// TIA Portal V20 export
FUNCTION_BLOCK "Simulation"   // FB50062, LAD
// stored: MemoryReserve 100, Namespace Unit1.Em7, SetENOAutomatically false
   VAR_INPUT
      simulation { ExternalAccessible := 'False'; ExternalVisible := 'False'; ExternalWritable := 'False'} : Bool;
   END_VAR
   VAR
      instActuator { ExternalAccessible := 'False'; ExternalVisible := 'False'; ExternalWritable := 'False'} : Array[0..19] of "LER_SimActuator";
   END_VAR
   VAR_TEMP   // added for the SCL form of the ladder/FBD networks
      _w1 : Bool;
      _w2 : Bool;
      _w3 : Bool;
      _w4 : Bool;
      _w5 : Bool;
      _w6 : Bool;
   END_VAR
BEGIN

REGION Network 1: Two Way Actuator
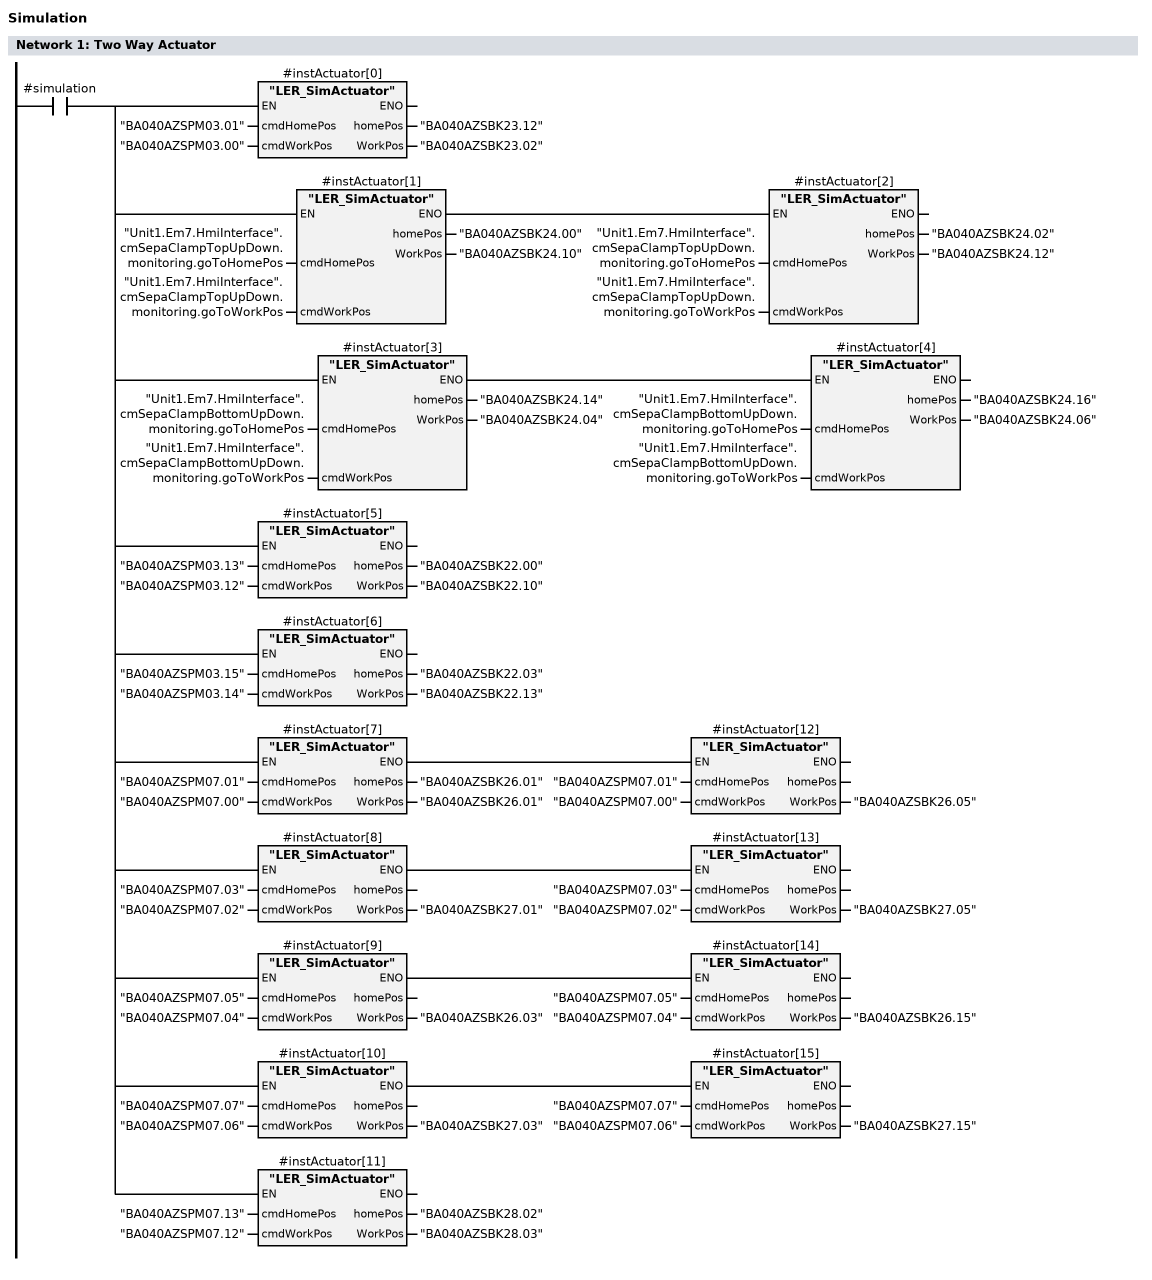
   RUNG wire#powerrail
      Contact( #simulation )
      wire#w1
      #instActuator[0](cmdHomePos := "BA040AZSPM03.01", cmdWorkPos := "BA040AZSPM03.00", homePos => "BA040AZSBK23.12", WorkPos => "BA040AZSBK23.02")
   END_RUNG
   RUNG wire#w1
      #instActuator[1](cmdHomePos := "Unit1.Em7.HmiInterface".cmSepaClampTopUpDown.monitoring.goToHomePos, cmdWorkPos := "Unit1.Em7.HmiInterface".cmSepaClampTopUpDown.monitoring.goToWorkPos, homePos => "BA040AZSBK24.00", WorkPos => "BA040AZSBK24.10")
      #instActuator[2](cmdHomePos := "Unit1.Em7.HmiInterface".cmSepaClampTopUpDown.monitoring.goToHomePos, cmdWorkPos := "Unit1.Em7.HmiInterface".cmSepaClampTopUpDown.monitoring.goToWorkPos, homePos => "BA040AZSBK24.02", WorkPos => "BA040AZSBK24.12")
   END_RUNG
   RUNG wire#w1
      #instActuator[3](cmdHomePos := "Unit1.Em7.HmiInterface".cmSepaClampBottomUpDown.monitoring.goToHomePos, cmdWorkPos := "Unit1.Em7.HmiInterface".cmSepaClampBottomUpDown.monitoring.goToWorkPos, homePos => "BA040AZSBK24.14", WorkPos => "BA040AZSBK24.04")
      #instActuator[4](cmdHomePos := "Unit1.Em7.HmiInterface".cmSepaClampBottomUpDown.monitoring.goToHomePos, cmdWorkPos := "Unit1.Em7.HmiInterface".cmSepaClampBottomUpDown.monitoring.goToWorkPos, homePos => "BA040AZSBK24.16", WorkPos => "BA040AZSBK24.06")
   END_RUNG
   RUNG wire#w1
      #instActuator[5](cmdHomePos := "BA040AZSPM03.13", cmdWorkPos := "BA040AZSPM03.12", homePos => "BA040AZSBK22.00", WorkPos => "BA040AZSBK22.10")
   END_RUNG
   RUNG wire#w1
      #instActuator[6](cmdHomePos := "BA040AZSPM03.15", cmdWorkPos := "BA040AZSPM03.14", homePos => "BA040AZSBK22.03", WorkPos => "BA040AZSBK22.13")
   END_RUNG
   RUNG wire#w1
      #instActuator[7](cmdHomePos := "BA040AZSPM07.01", cmdWorkPos := "BA040AZSPM07.00", homePos => "BA040AZSBK26.01", WorkPos => "BA040AZSBK26.01")
      #instActuator[12](cmdHomePos := "BA040AZSPM07.01", cmdWorkPos := "BA040AZSPM07.00", homePos =>, WorkPos => "BA040AZSBK26.05")
   END_RUNG
   RUNG wire#w1
      #instActuator[8](cmdHomePos := "BA040AZSPM07.03", cmdWorkPos := "BA040AZSPM07.02", homePos =>, WorkPos => "BA040AZSBK27.01")
      #instActuator[13](cmdHomePos := "BA040AZSPM07.03", cmdWorkPos := "BA040AZSPM07.02", homePos =>, WorkPos => "BA040AZSBK27.05")
   END_RUNG
   RUNG wire#w1
      #instActuator[9](cmdHomePos := "BA040AZSPM07.05", cmdWorkPos := "BA040AZSPM07.04", homePos =>, WorkPos => "BA040AZSBK26.03")
      #instActuator[14](cmdHomePos := "BA040AZSPM07.05", cmdWorkPos := "BA040AZSPM07.04", homePos =>, WorkPos => "BA040AZSBK26.15")
   END_RUNG
   RUNG wire#w1
      #instActuator[10](cmdHomePos := "BA040AZSPM07.07", cmdWorkPos := "BA040AZSPM07.06", homePos =>, WorkPos => "BA040AZSBK27.03")
      #instActuator[15](cmdHomePos := "BA040AZSPM07.07", cmdWorkPos := "BA040AZSPM07.06", homePos =>, WorkPos => "BA040AZSBK27.15")
   END_RUNG
   RUNG wire#w1
      #instActuator[11](cmdHomePos := "BA040AZSPM07.13", cmdWorkPos := "BA040AZSPM07.12", homePos => "BA040AZSBK28.02", WorkPos => "BA040AZSBK28.03")
   END_RUNG
   // the same network as SCL:
   IF #simulation THEN
       #instActuator[0](cmdHomePos := "BA040AZSPM03.01",   // "LER_SimActuator"
                        cmdWorkPos := "BA040AZSPM03.00",
                        homePos => "BA040AZSBK23.12",
                        WorkPos => "BA040AZSBK23.02");
   END_IF;
   #instActuator[1](EN := #simulation,   // "LER_SimActuator"
                    cmdHomePos := "Unit1.Em7.HmiInterface".cmSepaClampTopUpDown.monitoring.goToHomePos,
                    cmdWorkPos := "Unit1.Em7.HmiInterface".cmSepaClampTopUpDown.monitoring.goToWorkPos,
                    homePos => "BA040AZSBK24.00",
                    WorkPos => "BA040AZSBK24.10",
                    ENO => #_w1);
   IF #_w1 THEN
       #instActuator[2](cmdHomePos := "Unit1.Em7.HmiInterface".cmSepaClampTopUpDown.monitoring.goToHomePos,   // "LER_SimActuator"
                        cmdWorkPos := "Unit1.Em7.HmiInterface".cmSepaClampTopUpDown.monitoring.goToWorkPos,
                        homePos => "BA040AZSBK24.02",
                        WorkPos => "BA040AZSBK24.12");
   END_IF;
   #instActuator[3](EN := #simulation,   // "LER_SimActuator"
                    cmdHomePos := "Unit1.Em7.HmiInterface".cmSepaClampBottomUpDown.monitoring.goToHomePos,
                    cmdWorkPos := "Unit1.Em7.HmiInterface".cmSepaClampBottomUpDown.monitoring.goToWorkPos,
                    homePos => "BA040AZSBK24.14",
                    WorkPos => "BA040AZSBK24.04",
                    ENO => #_w2);
   IF #_w2 THEN
       #instActuator[4](cmdHomePos := "Unit1.Em7.HmiInterface".cmSepaClampBottomUpDown.monitoring.goToHomePos,   // "LER_SimActuator"
                        cmdWorkPos := "Unit1.Em7.HmiInterface".cmSepaClampBottomUpDown.monitoring.goToWorkPos,
                        homePos => "BA040AZSBK24.16",
                        WorkPos => "BA040AZSBK24.06");
   END_IF;
   IF #simulation THEN
       #instActuator[5](cmdHomePos := "BA040AZSPM03.13",   // "LER_SimActuator"
                        cmdWorkPos := "BA040AZSPM03.12",
                        homePos => "BA040AZSBK22.00",
                        WorkPos => "BA040AZSBK22.10");
       #instActuator[6](cmdHomePos := "BA040AZSPM03.15",   // "LER_SimActuator"
                        cmdWorkPos := "BA040AZSPM03.14",
                        homePos => "BA040AZSBK22.03",
                        WorkPos => "BA040AZSBK22.13");
   END_IF;
   #instActuator[7](EN := #simulation,   // "LER_SimActuator"
                    cmdHomePos := "BA040AZSPM07.01",
                    cmdWorkPos := "BA040AZSPM07.00",
                    homePos => "BA040AZSBK26.01",
                    WorkPos => "BA040AZSBK26.01",
                    ENO => #_w3);
   IF #_w3 THEN
       #instActuator[12](cmdHomePos := "BA040AZSPM07.01",   // "LER_SimActuator"
                         cmdWorkPos := "BA040AZSPM07.00",
                         WorkPos => "BA040AZSBK26.05");
   END_IF;
   #instActuator[8](EN := #simulation,   // "LER_SimActuator"
                    cmdHomePos := "BA040AZSPM07.03",
                    cmdWorkPos := "BA040AZSPM07.02",
                    WorkPos => "BA040AZSBK27.01",
                    ENO => #_w4);
   IF #_w4 THEN
       #instActuator[13](cmdHomePos := "BA040AZSPM07.03",   // "LER_SimActuator"
                         cmdWorkPos := "BA040AZSPM07.02",
                         WorkPos => "BA040AZSBK27.05");
   END_IF;
   #instActuator[9](EN := #simulation,   // "LER_SimActuator"
                    cmdHomePos := "BA040AZSPM07.05",
                    cmdWorkPos := "BA040AZSPM07.04",
                    WorkPos => "BA040AZSBK26.03",
                    ENO => #_w5);
   IF #_w5 THEN
       #instActuator[14](cmdHomePos := "BA040AZSPM07.05",   // "LER_SimActuator"
                         cmdWorkPos := "BA040AZSPM07.04",
                         WorkPos => "BA040AZSBK26.15");
   END_IF;
   #instActuator[10](EN := #simulation,   // "LER_SimActuator"
                     cmdHomePos := "BA040AZSPM07.07",
                     cmdWorkPos := "BA040AZSPM07.06",
                     WorkPos => "BA040AZSBK27.03",
                     ENO => #_w6);
   IF #_w6 THEN
       #instActuator[15](cmdHomePos := "BA040AZSPM07.07",   // "LER_SimActuator"
                         cmdWorkPos := "BA040AZSPM07.06",
                         WorkPos => "BA040AZSBK27.15");
   END_IF;
   IF #simulation THEN
       #instActuator[11](cmdHomePos := "BA040AZSPM07.13",   // "LER_SimActuator"
                         cmdWorkPos := "BA040AZSPM07.12",
                         homePos => "BA040AZSBK28.02",
                         WorkPos => "BA040AZSBK28.03");
   END_IF;
END_REGION
END_FUNCTION_BLOCK
